TYPE HB :
STRUCT
	HEARTBEAT		:BOOL	:= FALSE; //check in MQTTCOM to keep jog commands online
END_STRUCT
END_TYPE

(* stored: Version 1.1.0.1, ProductVersion 3.1.4026.18
   DUT HB: Id {2f72543e-9bd2-44cc-b81e-82fad39a7d1e} *)
